% RSLogix 500 project PLC_1_L5-1.RSS, saved by version 12.00.00.00 %
PROJECT "UNTITLED"    % processor: Bul.1763 MicroLogix 1100 Series B %

PROGRAM FILES
  LAD 2   4 rungs

DATA FILES
  O0 OUTPUT  5 elements
  I1 INPUT  6 elements
  S2 STATUS  66 elements
  B3 BINARY  1 elements
  T4 TIMER  1 elements
  C5 COUNTER  1 elements
  R6 CONTROL  1 elements
  N7 INTEGER  1 elements
  F8 FLOAT  1 elements

LADDER 2
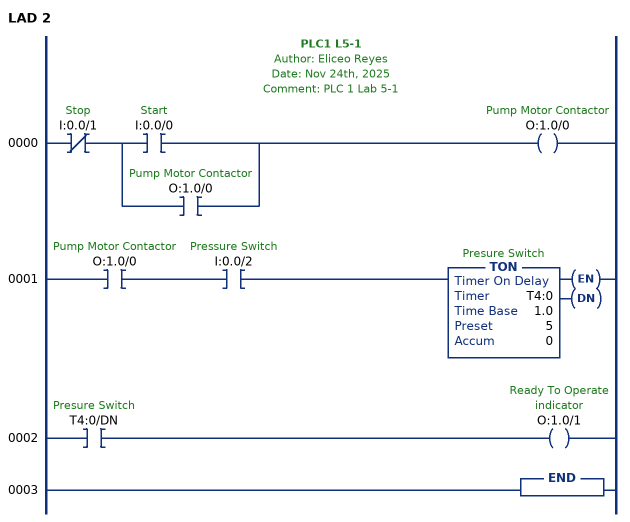
% Rung: 0 %
% TITLE: PLC1 L5-1 %
% Author: Eliceo Reyes
% Date: Nov 24th, 2025
% Comment: PLC 1 Lab 5-1 %
SOR XIO I:0.0/1 BST XIC I:0.0/0 NXB XIC O:1.0/0 BND OTE O:1.0/0 EOR
%   I:0.0/1  "Stop" %
%   I:0.0/0  "Start" %
%   O:1.0/0  "Pump Motor Contactor" %
% Rung: 1 %
SOR XIC O:1.0/0 XIC I:0.0/2 TON T4:0 1.0 5 0 EOR
%   O:1.0/0  "Pump Motor Contactor" %
%   I:0.0/2  "Pressure Switch" %
%   T4:0  "Presure Switch" %
% Rung: 2 %
SOR XIC T4:0/DN OTE O:1.0/1 EOR
%   T4:0  "Presure Switch" %
%   O:1.0/1  "Ready To Operate indicator" %
% Rung: 3 %
SOR END EOR

DATA TABLE (non-zero values as saved)
DATA T4
% .PRE .ACC %
% T4:0 % 5 0
